(* IEC 61131-3 sources: Laboratorijsko-busace-postrojenje/Libraries/adsWITS0, 3 files *)

(* ---- adsWITS0.typ ---- *)
(********************************************************************
 * COPYRIGHT --
 ********************************************************************
 * Library: adsWITS0
 * File: adsWITS0.typ
 * Author: fasch_f
 * Created: August 11, 2010
 ********************************************************************
 * Data types of library adsWITS0
 ********************************************************************)

TYPE
	RECORD_INFO_TYP : 	STRUCT
		recType : STRING[3];
		recNum : UINT := 0; (*actual number of records*)
		recSize : UINT := 0; (*record size in bytes*)
		wellIDSize : UINT := 0; (*size of the first record entry (Record-ID)*)
		pRecData : UDINT; (*pointer to record data*)
		recMaxSize : UINT := 0; (*maximum size of WITS-Record*)
		recActSize : UINT := 0; (*size of record with actual data*)
	END_STRUCT;
	DORECORD_INFO_TYP : 	STRUCT
		recType : STRING[3];
		recNum : UINT;
		recSize : UDINT;
		wellIDSize : UINT;
		pRecData : UDINT;
		ident : USINT;
	END_STRUCT;
END_TYPE

(* ---- adsWITS0.fun ---- *)
(********************************************************************
 * COPYRIGHT --
 ********************************************************************
 * Library: adsWITS0
 * File: adsWITS0.fun
 * Author: fasch_f
 * Created: August 11, 2010
 ********************************************************************
 * Functions and function blocks of library adsWITS0
 ********************************************************************)

FUNCTION witsInitRecordMin : UDINT (*function initialises a WITS Infotyp-Structure, without Well-Identifier-String*)
	VAR_INPUT
		RecType : STRING[3];
		pInfoStruct : UDINT;
		pDataArea : UDINT;
		AreaLen : UINT;
	END_VAR
END_FUNCTION

FUNCTION witsInitRecord : UDINT (*function initialises a WITS Infotyp-Structure*)
	VAR_INPUT
		RecType : STRING[3];
		pWellID : UDINT;
		pInfoStruct : UDINT;
		pDataArea : UDINT;
		AreaLen : UINT;
	END_VAR
END_FUNCTION

FUNCTION witsAddData : UDINT (*Adds data with ID and value to a WITS-Record*)
	VAR_INPUT
		pInfoStruct : UDINT;
		ItemID : STRING[3];
		pItemVal : UDINT;
	END_VAR
END_FUNCTION

FUNCTION witsUpdData : UDINT (*resets InfoStructure, so that data can updated by using witsAddData*)
	VAR_INPUT
		pInfoStruct : UDINT;
	END_VAR
END_FUNCTION

(* ---- adsWITS0.var ---- *)
(********************************************************************
 * COPYRIGHT --
 ********************************************************************
 * Library: adsWITS0
 * File: adsWITS0.var
 * Author: fasch_f
 * Created: August 11, 2010
 ********************************************************************
 * Constants of library adsWITS0
 ********************************************************************)
VAR CONSTANT
	WITS_PARERROR : UDINT := 10001;
	WITS_NOAREA : UDINT := 10002;
	WITS_RECORD_FULL : UDINT := 10003;
END_VAR
(*Record ID Constants*)
VAR CONSTANT
	WITS_REC_GENTIME : STRING[3] := '01';
	WITS_REC_DRILDEPTH : STRING[3] := '02';
END_VAR
(*Item ID Constants*)
VAR CONSTANT
	WITS_ITEM_WELLID : STRING[3] := '01';
	WITS_ITEM_DATE : STRING[3] := '05';
	WITS_ITEM_TIME : STRING[3] := '06';
	WITS_ITEM_BLOCKPOS : STRING[3] := '12';
	WITS_ITEM_RATEOFPEN : STRING[3] := '13';
	WITS_ITEM_ROTTORQUE_AVG : STRING[3] := '18';
	WITS_ITEM_ROTSPEED_AVG : STRING[3] := '20';
	WITS_ITEM_SPARE1 : STRING[3] := '41';
	WITS_ITEM_SPARE2 : STRING[3] := '42';
	WITS_ITEM_SPARE3 : STRING[3] := '43';
	WITS_ITEM_SPARE4 : STRING[3] := '44';
END_VAR
